(* PLC project Aufgabenserie2, Beckhoff Automation GmbH TwinCAT PLC Control 3.5.10.30 *)
(* stored: creationDateTime 2018-11-08T18:14:53.7227744, modificationDateTime 2018-11-08T18:14:53.7297742 *)

FUNCTION AdditionFunction : REAL
VAR_INPUT
	i_rValueA : REAL;
	i_rValueB : REAL;
END_VAR
VAR
END_VAR

            AdditionFunction := i_rValueA + i_rValueB;
          
END_FUNCTION
